{attribute 'qualified_only'}
{attribute 'strict'}
TYPE E_FutureExecutionState :
(
	idle := 0,
	init,
	wait_for_process,
	process,
	abort,
	quit,
	finish
);
END_TYPE

(* stored: Version 1.1.0.1, ProductVersion 3.1.4024.12
   DUT E_FutureExecutionState: Id {db307e80-41b8-4cda-abb3-bd9c8f7b3495} *)
